# EPICS autosave request: optics/opticsApp/Db/filterBladeNoSensor.req
$(P)$(R)Fi$(N):Enable
$(P)$(R)Fi$(N):Lock
$(P)$(R)Fi$(N):Thickness
$(P)$(R)Fi$(N):Material
